Staubli VAL3: StaubliUI.dtx

mdesc mNomSpeed
num nPanelLTopX
num nPanelLTopY
num nPanelWidthX
num nPanelLengthY
string sBuff
string sData
